FUNCTION_BLOCK FB_Properties
VAR_INPUT
END_VAR
VAR_OUTPUT
END_VAR
VAR
END_VAR

{attribute 'OPC.UA.DA.Property' := '1'}
{attribute 'monitoring' := 'call'}
PROPERTY MyProperty1 : BOOL
GET
END_GET
SET
END_SET
END_PROPERTY

END_FUNCTION_BLOCK

(* stored: Version 1.1.0.1, ProductVersion 3.1.4024.10
   POU FB_Properties: Id {52da11e9-c7f6-41cc-97e6-b578e0fee606}, SpecialFunc None
   Property MyProperty1: Id {6dab72ae-36ea-425b-901e-e597e4a770d1}
   Get Get: Id {1616f76b-00c7-4b3c-ace2-b501d1727482}
   Set Set: Id {98a1fda8-9f23-4b09-8692-aa674b2e6d7c} *)
